(* Logix 5000 project; controller cal1615 1756-L62 rev 20.11; software revision 20.05; part 30 of 81 *)
(* tags used below, declared in another part *)
   FAULT : BOOL;   // Fault AFI
   HMI : BOOL;   // AFI HMI
   p01r09_pb_global_reset : BOOL;   // System Modes PB: Global Fault Reset
   p13_ai_exhaust_amps : REAL;   // Zone 3 Analog Input Exhaust Fan Amps
   p13_ai_exhaust_hz : REAL;   // Zone 3 Analog Input Exhaust Fan HZ
   p13_ai_exhaust_pct : REAL;   // Zone 3 Analog Input Exhaust Fan PCT
   p13_ai_exhaust_rpm : REAL;   // Zone 3 Analog Input Exhaust Fan RPM
   p13_ai_recirc_amps : REAL;   // Zone 3 Analog Input Recirc Fan Amps
   p13_ai_recirc_hz : REAL;   // Zone 3 Analog Input Supply Fan HZ
   p13_ai_recirc_pct : REAL;   // Zone 3 Analog Input Recirc Fan PCT
   p13_ai_recirc_rpm : REAL;   // Zone 3 Analog Input Recirc Fan RPM
   p13_ai_tc01 : REAL;   // Zone 3 Analog Input Control Thermocouple 1
   p13_ai_tc02 : REAL;   // Zone 3 Analog Input Control Thermocouple 2
   p13_ao_cv : REAL;   // Zone 3 Analog Output Control Valve
   p13_ao_exhaust_selected_speed : REAL;   // Zone 3 Analog Output Exhaust Fan VFD Selected Speed
   p13_ao_recirc_selected_speed : REAL;   // Zone 3 Analog Output Recirc Fan VFD Selected Speed
   p13_di_recirc : acs800_di_normal;   // Zone 3 Digital Inputs Recirc Fan
   p13_dint_to_hmi : DINT[16];   // Zone 3 Temperature Control VFDs On
   p13_param_fast_to_soak : REAL;   // Zone 3 Parameter Fast to Soak Control
   p13_param_lfl_hhl : REAL;   // Zone 3 Parameter High High Lower Flash Limit
   p13_param_lfl_hl : REAL;   // Zone 3 Parameter High LFL Limit
   p13_param_pid1_ff : REAL;   // Zone 3 Parameter Fast PID Bias
   p13_param_pid1_kd : REAL;   // Zone 3 Parameter Fast PID Derivative Gain
   p13_param_pid1_ki : REAL;   // Zone 3 Parameter Fast PID Integral Gain
   p13_param_pid1_kp : REAL;   // Zone 3 Parameter Fast PID Proportional Gain
   p13_param_pid2_ff : REAL;   // Zone 3 Parameter Auto PID Bias
   p13_param_pid2_kd : REAL;   // Zone 3 Parameter Auto PID Derivative Gain
   p13_param_pid2_ki : REAL;   // Zone 3 Parameter Auto PID Integral Gain
   p13_param_pid2_kp : REAL;   // Zone 3 Parameter Auto PID Proportional Gain
   p13_param_shutdown_temp : REAL;   // Zone 3 Parameter Zone Shutdown Temperature
   p13_param_soak_to_fast : REAL;   // Zone 3 Parameter Soak to Fast Control
   p13_param_tc01_dev : REAL;   // Zone 3 Parameter Oven Temperature Deviation from Setpoint
   p13_param_tc01_hl : REAL;   // Zone 3 Parameter Process Air High Limit
   p13_param_tc01z : REAL;   // Zone 3 Parameter Process Temperature Zero Offset
   p13_param_tc02z : REAL;   // Zone 3 Parameter SupplyTemperature Zero Offset
   p13_param_zone_pressure : REAL;   // Zone 3 Parameter High Pressure LImit
   p13_real_to_hmi : REAL[112];   // Zone 3 Real to HMI
   p13r01 : routine;   // Zone 3 Main
   p13r05 : routine;   // Zone 3 Dint to HMI
   p13r05_recirc_status : DINT;
   p13r05_timer_fault : TIMER[4];   // Zone 3 Dint to HMI Fault Delay
   p13r05_timer_warning : TIMER[4];   // Zone 3 Dint to HMI Warning Delay
   p13r06 : routine;   // Zone 3 Real to HMI
   p13r06_timer_fault : TIMER[4];   // Zone 3 Real to HMI Fault Delay
   p13r06_timer_warning : TIMER[4];   // Zone 3 Real to HMI Warning Delay
   p13r07 : routine;   // Zone 3 Alarms
   p13r07_timer_fault : TIMER[4];   // Zone 3 Alarms Fault Delay
   p13r07_timer_warning : TIMER[4];   // Zone 3 Alarms Warning Delay
   p13r08 : routine;   // Zone 3 Warnings
   p13r08_timer_fault : TIMER[4];   // Zone 3 Warnings Fault Delay
   p13r08_timer_warning : TIMER[4];   // Zone 3 Warnings Warning Delay
   p13r20 : routine;   // Zone 3 Temp Sequence
   p13r30 : routine;   // Zone 3 Temperature Control
   p13r30_cv_man_sp : REAL;   // Zone 3 Temperature Control Manual Heat Control Valve Setpoint
   p13r30_pid_temp_pv : REAL;   // Zone 3 Temperature Control PID Process Value
   p13r30_pid_temp_sp : REAL;   // Zone 3 Temperature Control PID Temperature Control Setpoint
   p13r31 : routine;   // Zone 3 Exhaust VFD
   p13r32 : routine;   // Zone 3 Recirc VFD
   p13r32_vfd_stopped : BOOL;   // Zone 3 Recirc VFD VFD Stopped
(* P13_Zone_3, continued *)

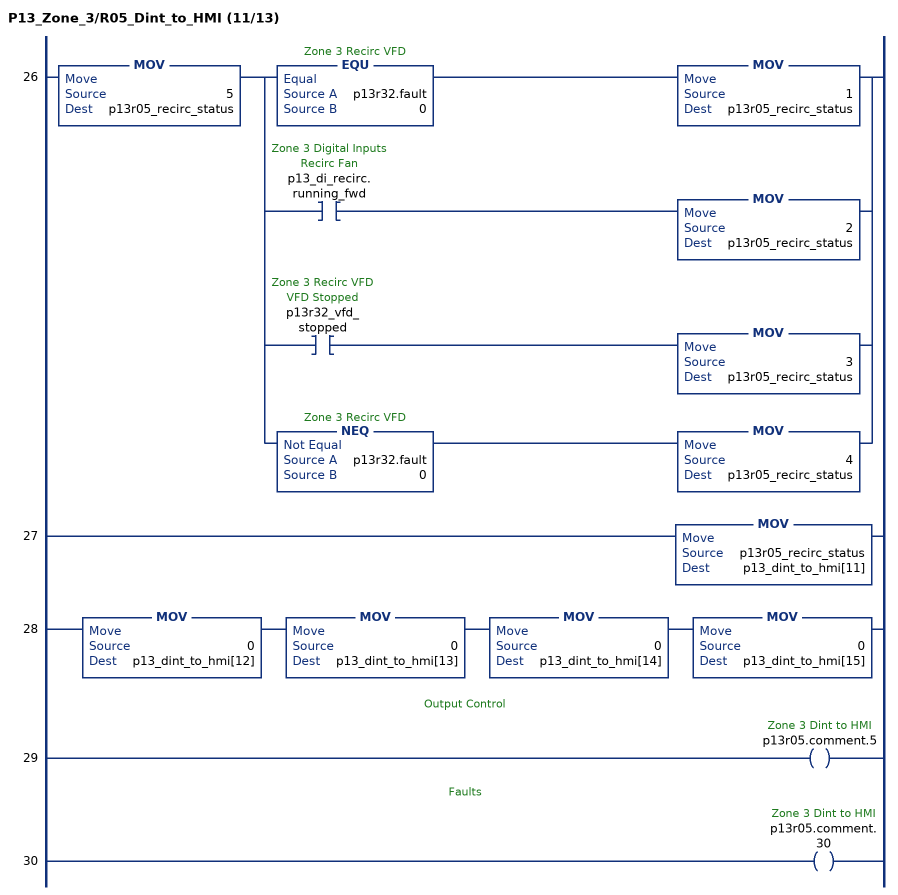
   [picture p524: P13_Zone_3/R05_Dint_to_HMI rungs 26-30]
   26: MOV(5,p13r05_recirc_status)[EQU(p13r32.fault,0) MOV(1,p13r05_recirc_status) ,XIC(p13_di_recirc.running_fwd) MOV(2,p13r05_recirc_status) ,XIC(p13r32_vfd_stopped) MOV(3,p13r05_recirc_status) ,NEQ(p13r32.fault,0) MOV(4,p13r05_recirc_status) ];
   27: MOV(p13r05_recirc_status,p13_dint_to_hmi[11]);
   28: MOV(0,p13_dint_to_hmi[12])MOV(0,p13_dint_to_hmi[13])MOV(0,p13_dint_to_hmi[14])MOV(0,p13_dint_to_hmi[15]);
   // Output Control
   29: OTE(p13r05.comment.5);
   // Faults
   30: OTE(p13r05.comment.30);
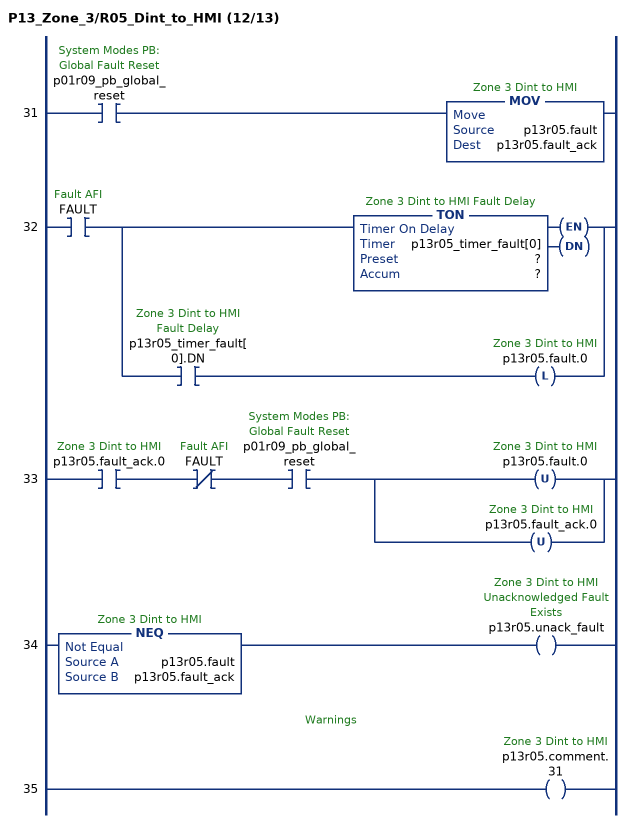
   31: XIC(p01r09_pb_global_reset)MOV(p13r05.fault,p13r05.fault_ack);
   32: XIC(FAULT)[TON(p13r05_timer_fault[0],?,?) ,XIC(p13r05_timer_fault[0].DN) OTL(p13r05.fault.0) ];
   33: XIC(p13r05.fault_ack.0)XIO(FAULT)XIC(p01r09_pb_global_reset)[OTU(p13r05.fault.0) ,OTU(p13r05.fault_ack.0) ];
   34: NEQ(p13r05.fault,p13r05.fault_ack)OTE(p13r05.unack_fault);
   // Warnings
   35: OTE(p13r05.comment.31);
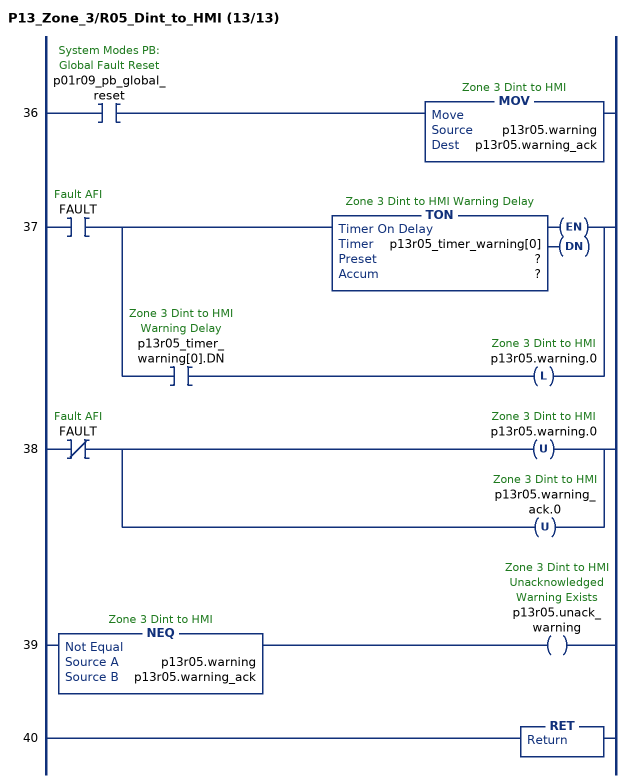
   36: XIC(p01r09_pb_global_reset)MOV(p13r05.warning,p13r05.warning_ack);
   37: XIC(FAULT)[TON(p13r05_timer_warning[0],?,?) ,XIC(p13r05_timer_warning[0].DN) OTL(p13r05.warning.0) ];
   38: XIO(FAULT)[OTU(p13r05.warning.0) ,OTU(p13r05.warning_ack.0) ];
   39: NEQ(p13r05.warning,p13r05.warning_ack)OTE(p13r05.unack_warning);
   40: RET();
END_ROUTINE

ROUTINE R06_Real_to_HMI   (* ladder *)
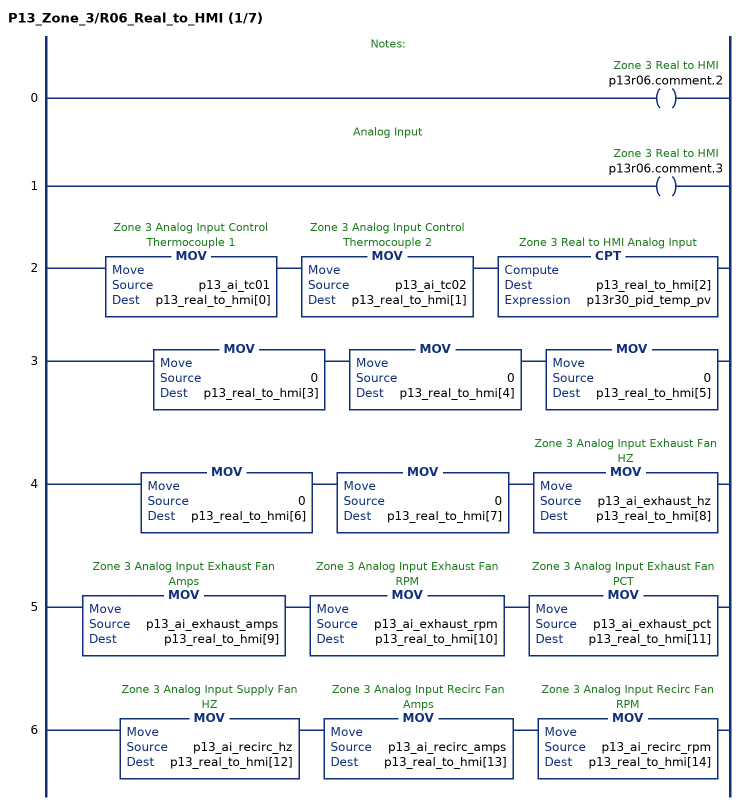
   // Notes:
   0: OTE(p13r06.comment.2);
   // Analog Input
   1: OTE(p13r06.comment.3);
   2: MOV(p13_ai_tc01,p13_real_to_hmi[0])MOV(p13_ai_tc02,p13_real_to_hmi[1])CPT(p13_real_to_hmi[2],p13r30_pid_temp_pv);
   3: MOV(0,p13_real_to_hmi[3])MOV(0,p13_real_to_hmi[4])MOV(0,p13_real_to_hmi[5]);
   4: MOV(0,p13_real_to_hmi[6])MOV(0,p13_real_to_hmi[7])MOV(p13_ai_exhaust_hz,p13_real_to_hmi[8]);
   5: MOV(p13_ai_exhaust_amps,p13_real_to_hmi[9])MOV(p13_ai_exhaust_rpm,p13_real_to_hmi[10])MOV(p13_ai_exhaust_pct,p13_real_to_hmi[11]);
   6: MOV(p13_ai_recirc_hz,p13_real_to_hmi[12])MOV(p13_ai_recirc_amps,p13_real_to_hmi[13])MOV(p13_ai_recirc_rpm,p13_real_to_hmi[14]);
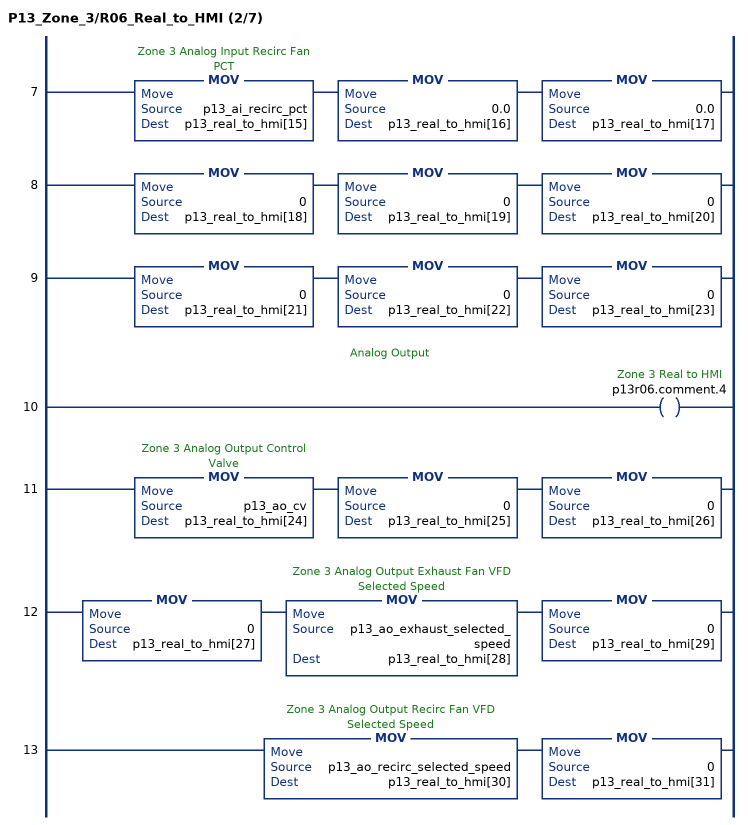
   7: MOV(p13_ai_recirc_pct,p13_real_to_hmi[15])MOV(0.0,p13_real_to_hmi[16])MOV(0.0,p13_real_to_hmi[17]);
   8: MOV(0,p13_real_to_hmi[18])MOV(0,p13_real_to_hmi[19])MOV(0,p13_real_to_hmi[20]);
   9: MOV(0,p13_real_to_hmi[21])MOV(0,p13_real_to_hmi[22])MOV(0,p13_real_to_hmi[23]);
   // Analog Output
   10: OTE(p13r06.comment.4);
   11: MOV(p13_ao_cv,p13_real_to_hmi[24])MOV(0,p13_real_to_hmi[25])MOV(0,p13_real_to_hmi[26]);
   12: MOV(0,p13_real_to_hmi[27])MOV(p13_ao_exhaust_selected_speed,p13_real_to_hmi[28])MOV(0,p13_real_to_hmi[29]);
   13: MOV(p13_ao_recirc_selected_speed,p13_real_to_hmi[30])MOV(0,p13_real_to_hmi[31]);
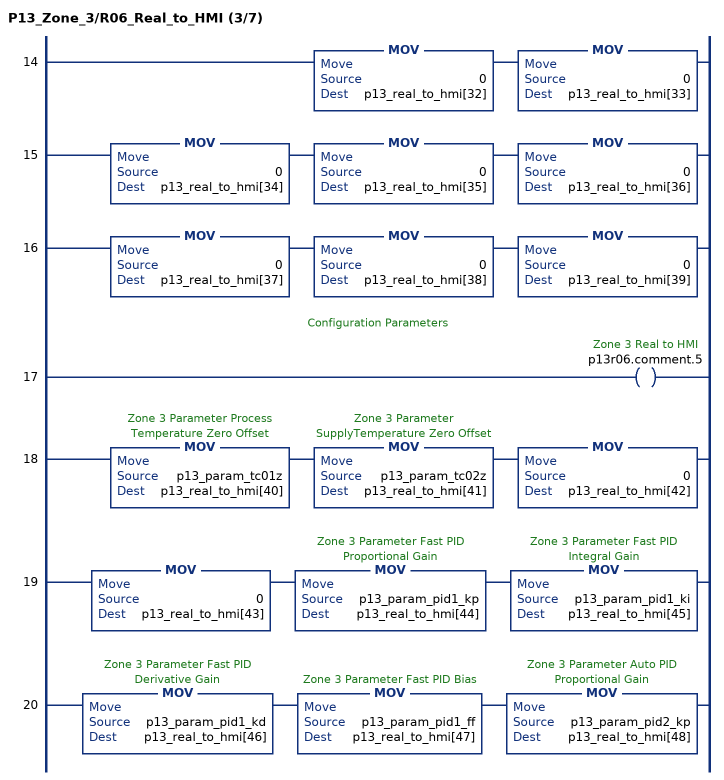
   14: MOV(0,p13_real_to_hmi[32])MOV(0,p13_real_to_hmi[33]);
   15: MOV(0,p13_real_to_hmi[34])MOV(0,p13_real_to_hmi[35])MOV(0,p13_real_to_hmi[36]);
   16: MOV(0,p13_real_to_hmi[37])MOV(0,p13_real_to_hmi[38])MOV(0,p13_real_to_hmi[39]);
   // Configuration Parameters
   17: OTE(p13r06.comment.5);
   18: MOV(p13_param_tc01z,p13_real_to_hmi[40])MOV(p13_param_tc02z,p13_real_to_hmi[41])MOV(0,p13_real_to_hmi[42]);
   19: MOV(0,p13_real_to_hmi[43])MOV(p13_param_pid1_kp,p13_real_to_hmi[44])MOV(p13_param_pid1_ki,p13_real_to_hmi[45]);
   20: MOV(p13_param_pid1_kd,p13_real_to_hmi[46])MOV(p13_param_pid1_ff,p13_real_to_hmi[47])MOV(p13_param_pid2_kp,p13_real_to_hmi[48]);
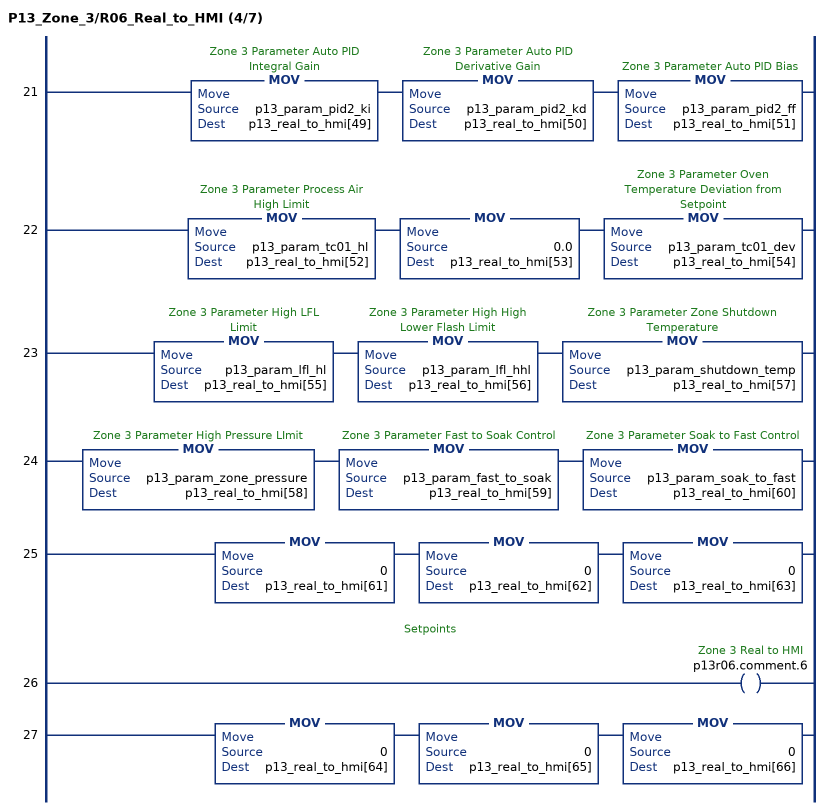
   21: MOV(p13_param_pid2_ki,p13_real_to_hmi[49])MOV(p13_param_pid2_kd,p13_real_to_hmi[50])MOV(p13_param_pid2_ff,p13_real_to_hmi[51]);
   22: MOV(p13_param_tc01_hl,p13_real_to_hmi[52])MOV(0.0,p13_real_to_hmi[53])MOV(p13_param_tc01_dev,p13_real_to_hmi[54]);
   23: MOV(p13_param_lfl_hl,p13_real_to_hmi[55])MOV(p13_param_lfl_hhl,p13_real_to_hmi[56])MOV(p13_param_shutdown_temp,p13_real_to_hmi[57]);
   24: MOV(p13_param_zone_pressure,p13_real_to_hmi[58])MOV(p13_param_fast_to_soak,p13_real_to_hmi[59])MOV(p13_param_soak_to_fast,p13_real_to_hmi[60]);
   25: MOV(0,p13_real_to_hmi[61])MOV(0,p13_real_to_hmi[62])MOV(0,p13_real_to_hmi[63]);
   // Setpoints
   26: OTE(p13r06.comment.6);
   27: MOV(0,p13_real_to_hmi[64])MOV(0,p13_real_to_hmi[65])MOV(0,p13_real_to_hmi[66]);
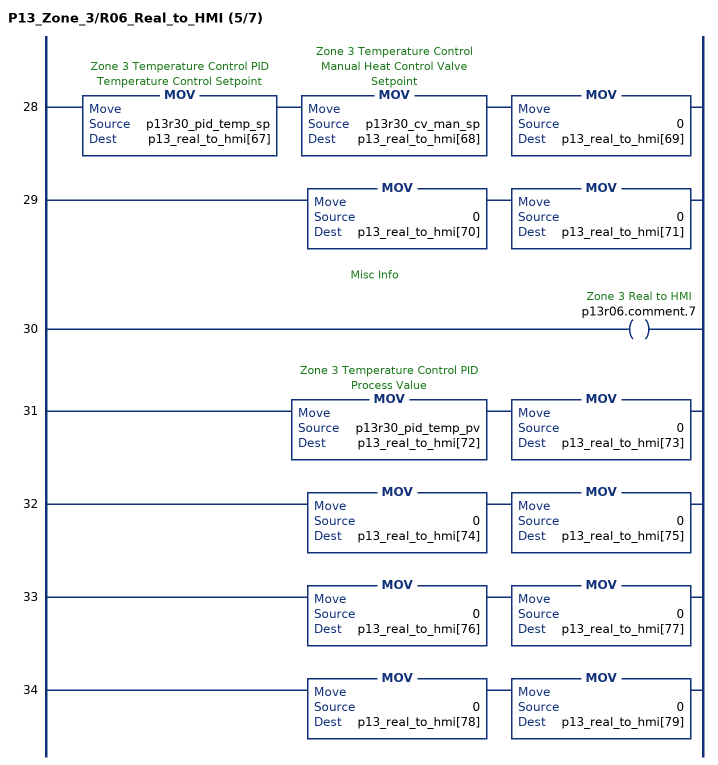
   28: MOV(p13r30_pid_temp_sp,p13_real_to_hmi[67])MOV(p13r30_cv_man_sp,p13_real_to_hmi[68])MOV(0,p13_real_to_hmi[69]);
   29: MOV(0,p13_real_to_hmi[70])MOV(0,p13_real_to_hmi[71]);
   // Misc Info
   30: OTE(p13r06.comment.7);
   31: MOV(p13r30_pid_temp_pv,p13_real_to_hmi[72])MOV(0,p13_real_to_hmi[73]);
   32: MOV(0,p13_real_to_hmi[74])MOV(0,p13_real_to_hmi[75]);
   33: MOV(0,p13_real_to_hmi[76])MOV(0,p13_real_to_hmi[77]);
   34: MOV(0,p13_real_to_hmi[78])MOV(0,p13_real_to_hmi[79]);
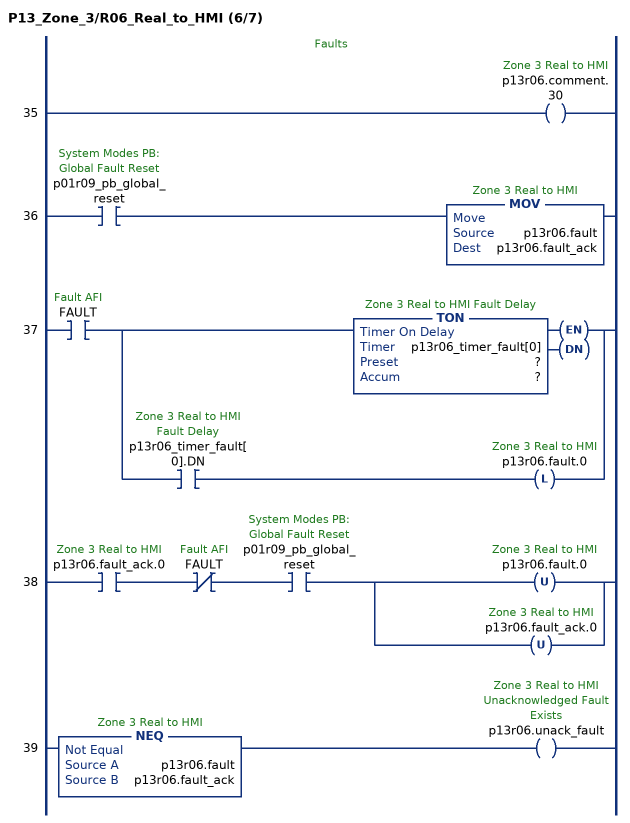
   // Faults
   35: OTE(p13r06.comment.30);
   36: XIC(p01r09_pb_global_reset)MOV(p13r06.fault,p13r06.fault_ack);
   37: XIC(FAULT)[TON(p13r06_timer_fault[0],?,?) ,XIC(p13r06_timer_fault[0].DN) OTL(p13r06.fault.0) ];
   38: XIC(p13r06.fault_ack.0)XIO(FAULT)XIC(p01r09_pb_global_reset)[OTU(p13r06.fault.0) ,OTU(p13r06.fault_ack.0) ];
   39: NEQ(p13r06.fault,p13r06.fault_ack)OTE(p13r06.unack_fault);
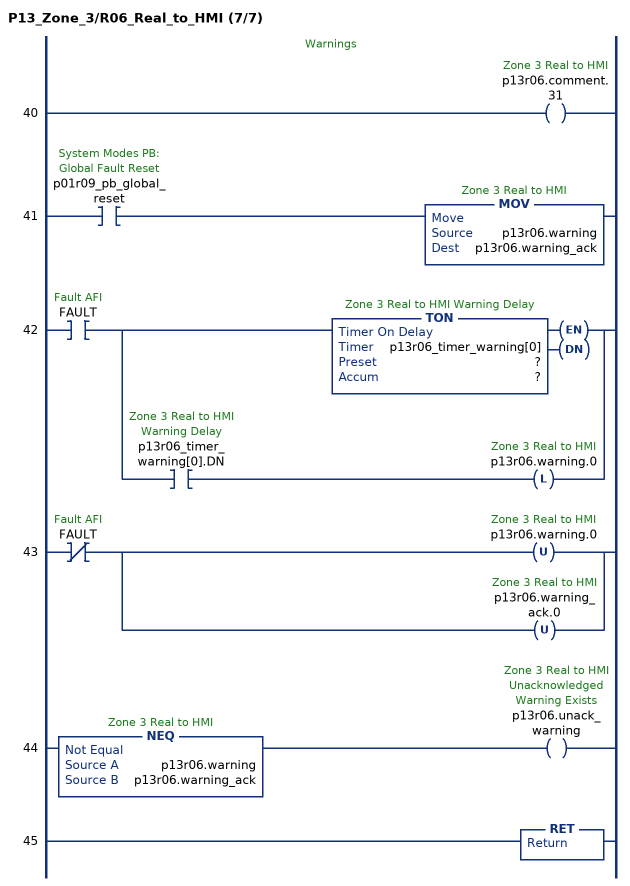
   // Warnings
   40: OTE(p13r06.comment.31);
   41: XIC(p01r09_pb_global_reset)MOV(p13r06.warning,p13r06.warning_ack);
   42: XIC(FAULT)[TON(p13r06_timer_warning[0],?,?) ,XIC(p13r06_timer_warning[0].DN) OTL(p13r06.warning.0) ];
   43: XIO(FAULT)[OTU(p13r06.warning.0) ,OTU(p13r06.warning_ack.0) ];
   44: NEQ(p13r06.warning,p13r06.warning_ack)OTE(p13r06.unack_warning);
   45: RET();
END_ROUTINE

ROUTINE R07_Alarms   (* ladder *)
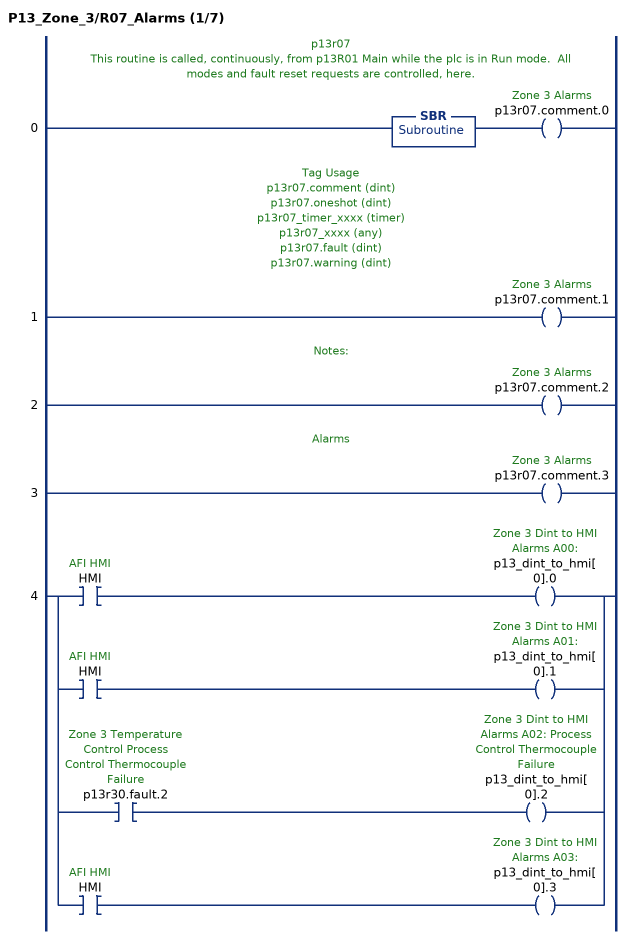
   // p13r07
   // This routine is called, continuously, from p13R01 Main while the plc is in Run mode.  All modes and fault reset requests are controlled, here.
   0: SBR()OTE(p13r07.comment.0);
   // Tag Usage
   // p13r07.comment (dint)
   // p13r07.oneshot (dint)
   // p13r07_timer_xxxx (timer)
   // p13r07_xxxx (any)
   // p13r07.fault (dint)
   // p13r07.warning (dint)
   1: OTE(p13r07.comment.1);
   // Notes:
   2: OTE(p13r07.comment.2);
   // Alarms
   3: OTE(p13r07.comment.3);
   4: [XIC(HMI) OTE(p13_dint_to_hmi[0].0) ,XIC(HMI) OTE(p13_dint_to_hmi[0].1) ,XIC(p13r30.fault.2) OTE(p13_dint_to_hmi[0].2) ,XIC(HMI) OTE(p13_dint_to_hmi[0].3) ];
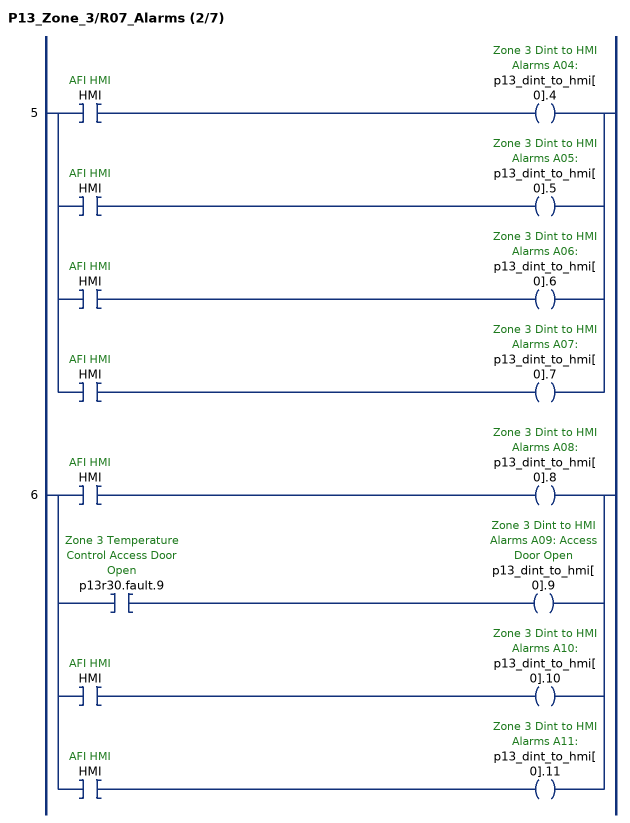
   5: [XIC(HMI) OTE(p13_dint_to_hmi[0].4) ,XIC(HMI) OTE(p13_dint_to_hmi[0].5) ,XIC(HMI) OTE(p13_dint_to_hmi[0].6) ,XIC(HMI) OTE(p13_dint_to_hmi[0].7) ];
   6: [XIC(HMI) OTE(p13_dint_to_hmi[0].8) ,XIC(p13r30.fault.9) OTE(p13_dint_to_hmi[0].9) ,XIC(HMI) OTE(p13_dint_to_hmi[0].10) ,XIC(HMI) OTE(p13_dint_to_hmi[0].11) ];
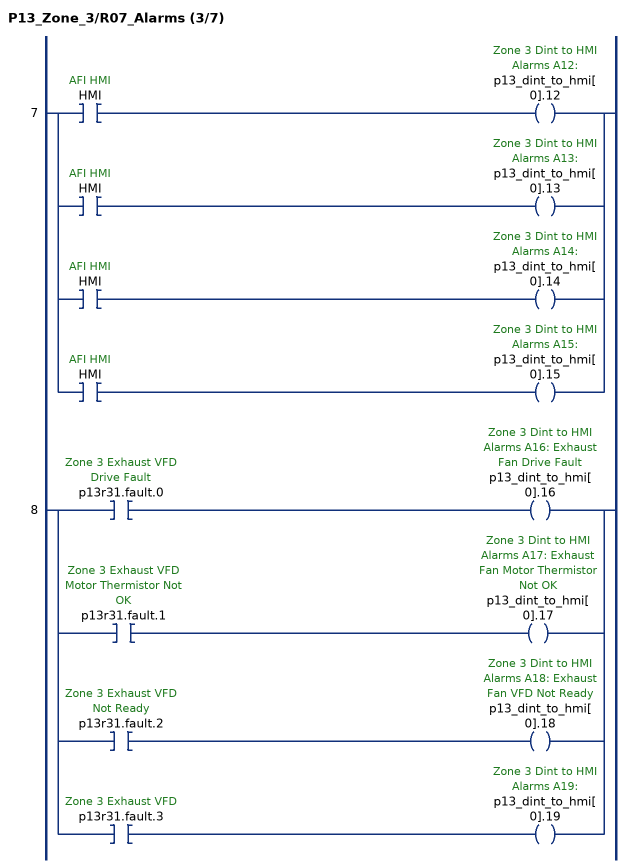
   7: [XIC(HMI) OTE(p13_dint_to_hmi[0].12) ,XIC(HMI) OTE(p13_dint_to_hmi[0].13) ,XIC(HMI) OTE(p13_dint_to_hmi[0].14) ,XIC(HMI) OTE(p13_dint_to_hmi[0].15) ];
   8: [XIC(p13r31.fault.0) OTE(p13_dint_to_hmi[0].16) ,XIC(p13r31.fault.1) OTE(p13_dint_to_hmi[0].17) ,XIC(p13r31.fault.2) OTE(p13_dint_to_hmi[0].18) ,XIC(p13r31.fault.3) OTE(p13_dint_to_hmi[0].19) ];
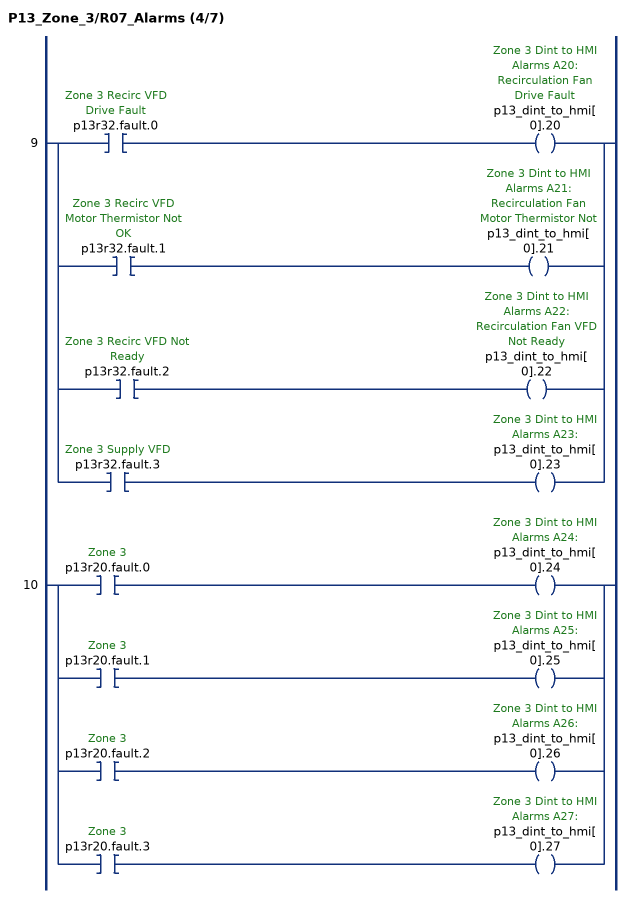
   9: [XIC(p13r32.fault.0) OTE(p13_dint_to_hmi[0].20) ,XIC(p13r32.fault.1) OTE(p13_dint_to_hmi[0].21) ,XIC(p13r32.fault.2) OTE(p13_dint_to_hmi[0].22) ,XIC(p13r32.fault.3) OTE(p13_dint_to_hmi[0].23) ];
   10: [XIC(p13r20.fault.0) OTE(p13_dint_to_hmi[0].24) ,XIC(p13r20.fault.1) OTE(p13_dint_to_hmi[0].25) ,XIC(p13r20.fault.2) OTE(p13_dint_to_hmi[0].26) ,XIC(p13r20.fault.3) OTE(p13_dint_to_hmi[0].27) ];
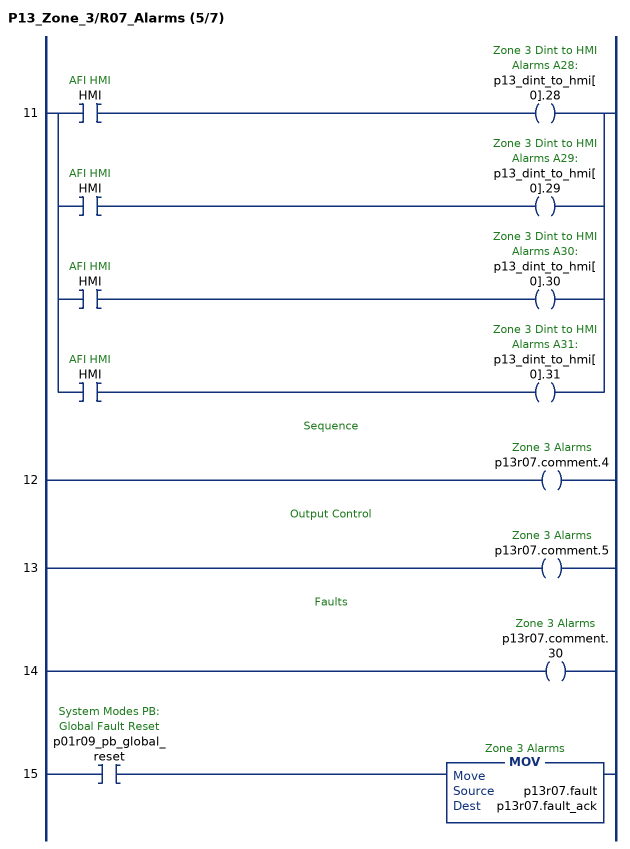
   11: [XIC(HMI) OTE(p13_dint_to_hmi[0].28) ,XIC(HMI) OTE(p13_dint_to_hmi[0].29) ,XIC(HMI) OTE(p13_dint_to_hmi[0].30) ,XIC(HMI) OTE(p13_dint_to_hmi[0].31) ];
   // Sequence
   12: OTE(p13r07.comment.4);
   // Output Control
   13: OTE(p13r07.comment.5);
   // Faults
   14: OTE(p13r07.comment.30);
   15: XIC(p01r09_pb_global_reset)MOV(p13r07.fault,p13r07.fault_ack);
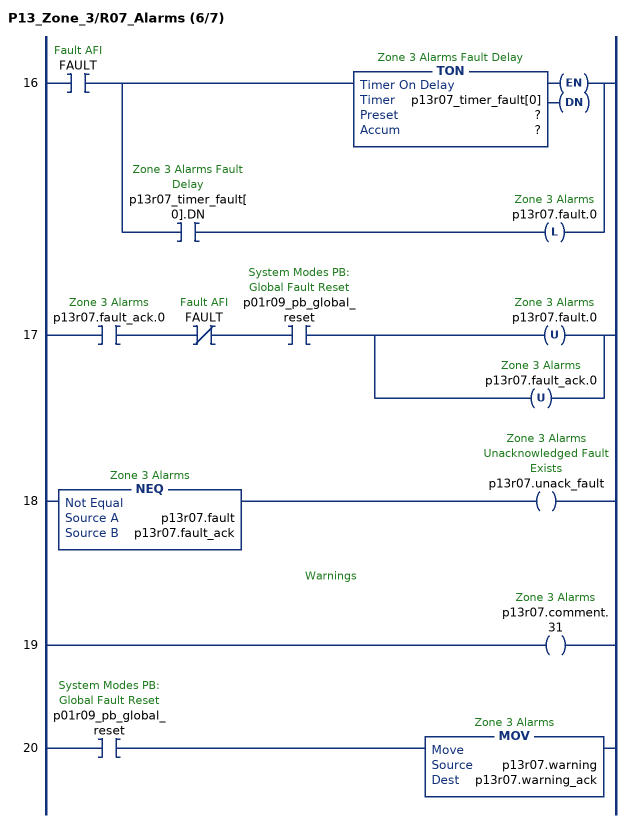
   16: XIC(FAULT)[TON(p13r07_timer_fault[0],?,?) ,XIC(p13r07_timer_fault[0].DN) OTL(p13r07.fault.0) ];
   17: XIC(p13r07.fault_ack.0)XIO(FAULT)XIC(p01r09_pb_global_reset)[OTU(p13r07.fault.0) ,OTU(p13r07.fault_ack.0) ];
   18: NEQ(p13r07.fault,p13r07.fault_ack)OTE(p13r07.unack_fault);
   // Warnings
   19: OTE(p13r07.comment.31);
   20: XIC(p01r09_pb_global_reset)MOV(p13r07.warning,p13r07.warning_ack);
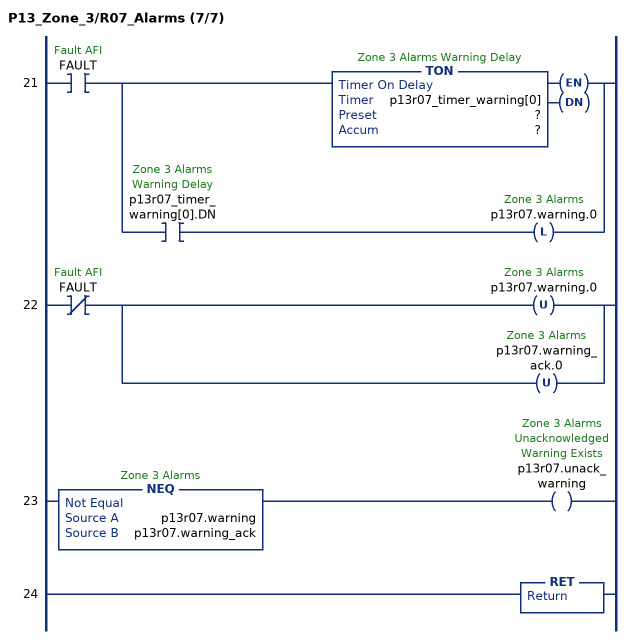
   21: XIC(FAULT)[TON(p13r07_timer_warning[0],?,?) ,XIC(p13r07_timer_warning[0].DN) OTL(p13r07.warning.0) ];
   22: XIO(FAULT)[OTU(p13r07.warning.0) ,OTU(p13r07.warning_ack.0) ];
   23: NEQ(p13r07.warning,p13r07.warning_ack)OTE(p13r07.unack_warning);
   24: RET();
END_ROUTINE

ROUTINE R08_Warnings   (* ladder *)
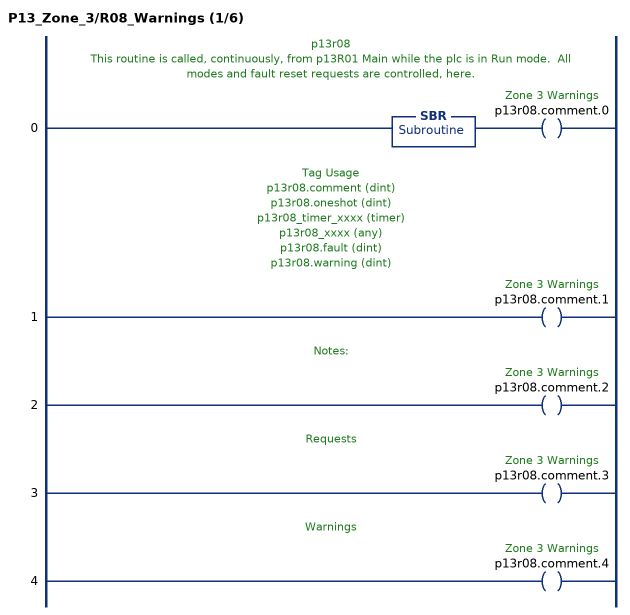
   // p13r08
   // This routine is called, continuously, from p13R01 Main while the plc is in Run mode.  All modes and fault reset requests are controlled, here.
   0: SBR()OTE(p13r08.comment.0);
   // Tag Usage
   // p13r08.comment (dint)
   // p13r08.oneshot (dint)
   // p13r08_timer_xxxx (timer)
   // p13r08_xxxx (any)
   // p13r08.fault (dint)
   // p13r08.warning (dint)
   1: OTE(p13r08.comment.1);
   // Notes:
   2: OTE(p13r08.comment.2);
   // Requests
   3: OTE(p13r08.comment.3);
   // Warnings
   4: OTE(p13r08.comment.4);
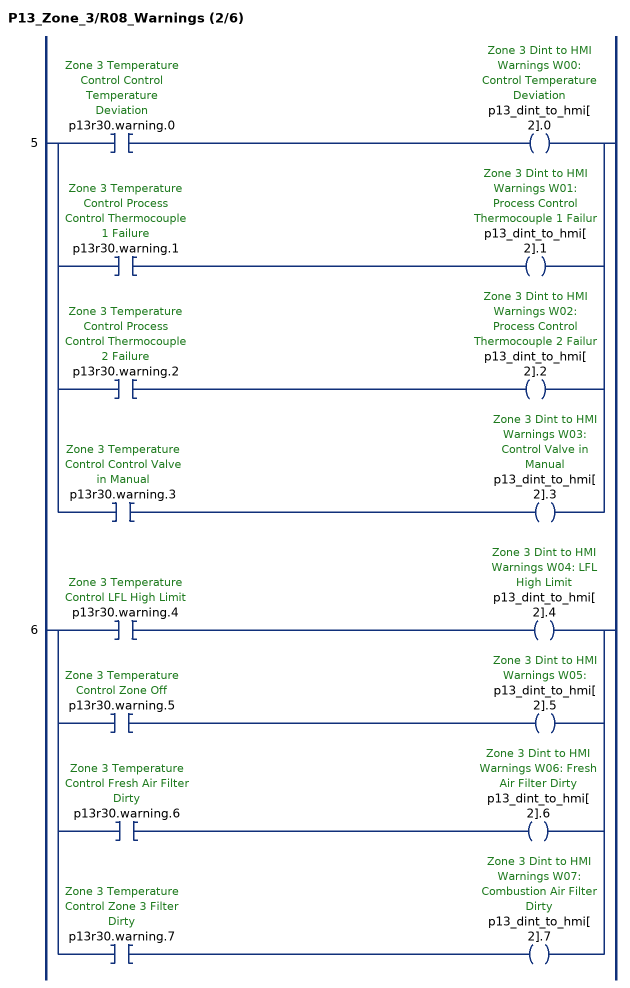
   5: [XIC(p13r30.warning.0) OTE(p13_dint_to_hmi[2].0) ,XIC(p13r30.warning.1) OTE(p13_dint_to_hmi[2].1) ,XIC(p13r30.warning.2) OTE(p13_dint_to_hmi[2].2) ,XIC(p13r30.warning.3) OTE(p13_dint_to_hmi[2].3) ];
   6: [XIC(p13r30.warning.4) OTE(p13_dint_to_hmi[2].4) ,XIC(p13r30.warning.5) OTE(p13_dint_to_hmi[2].5) ,XIC(p13r30.warning.6) OTE(p13_dint_to_hmi[2].6) ,XIC(p13r30.warning.7) OTE(p13_dint_to_hmi[2].7) ];
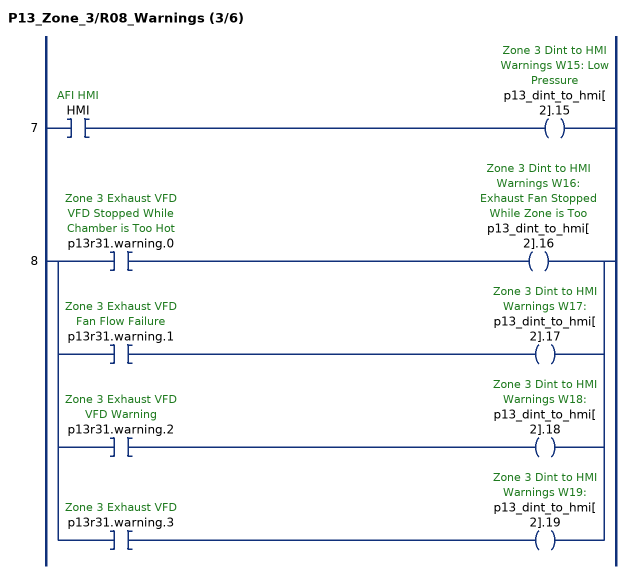
   7: XIC(HMI)OTE(p13_dint_to_hmi[2].15);
   8: [XIC(p13r31.warning.0) OTE(p13_dint_to_hmi[2].16) ,XIC(p13r31.warning.1) OTE(p13_dint_to_hmi[2].17) ,XIC(p13r31.warning.2) OTE(p13_dint_to_hmi[2].18) ,XIC(p13r31.warning.3) OTE(p13_dint_to_hmi[2].19) ];
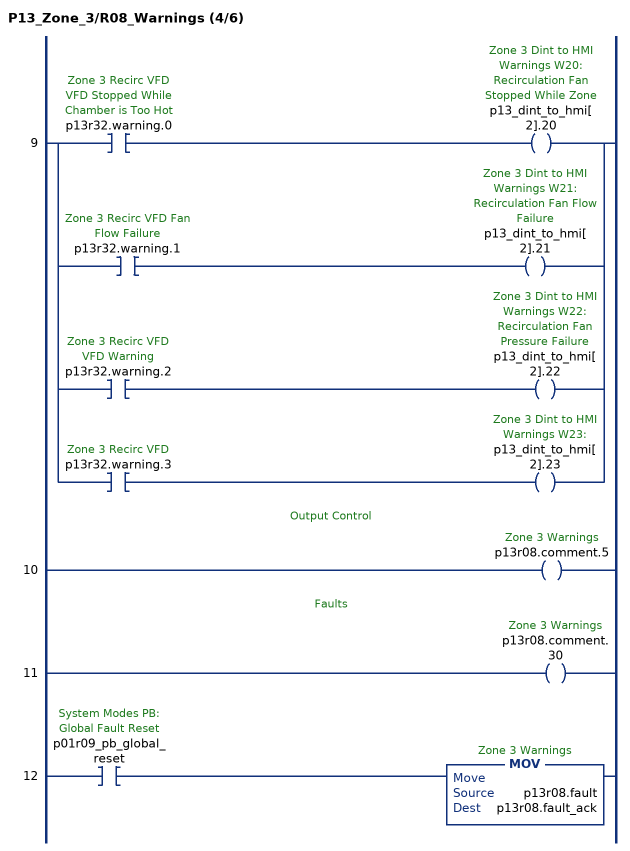
   9: [XIC(p13r32.warning.0) OTE(p13_dint_to_hmi[2].20) ,XIC(p13r32.warning.1) OTE(p13_dint_to_hmi[2].21) ,XIC(p13r32.warning.2) OTE(p13_dint_to_hmi[2].22) ,XIC(p13r32.warning.3) OTE(p13_dint_to_hmi[2].23) ];
   // Output Control
   10: OTE(p13r08.comment.5);
   // Faults
   11: OTE(p13r08.comment.30);
   12: XIC(p01r09_pb_global_reset)MOV(p13r08.fault,p13r08.fault_ack);
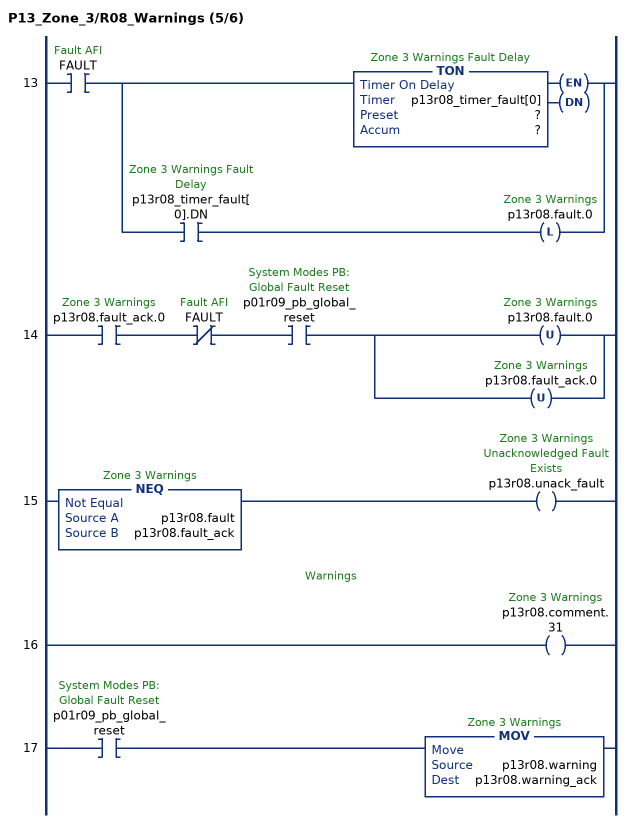
   13: XIC(FAULT)[TON(p13r08_timer_fault[0],?,?) ,XIC(p13r08_timer_fault[0].DN) OTL(p13r08.fault.0) ];
   14: XIC(p13r08.fault_ack.0)XIO(FAULT)XIC(p01r09_pb_global_reset)[OTU(p13r08.fault.0) ,OTU(p13r08.fault_ack.0) ];
   15: NEQ(p13r08.fault,p13r08.fault_ack)OTE(p13r08.unack_fault);
   // Warnings
   16: OTE(p13r08.comment.31);
   17: XIC(p01r09_pb_global_reset)MOV(p13r08.warning,p13r08.warning_ack);
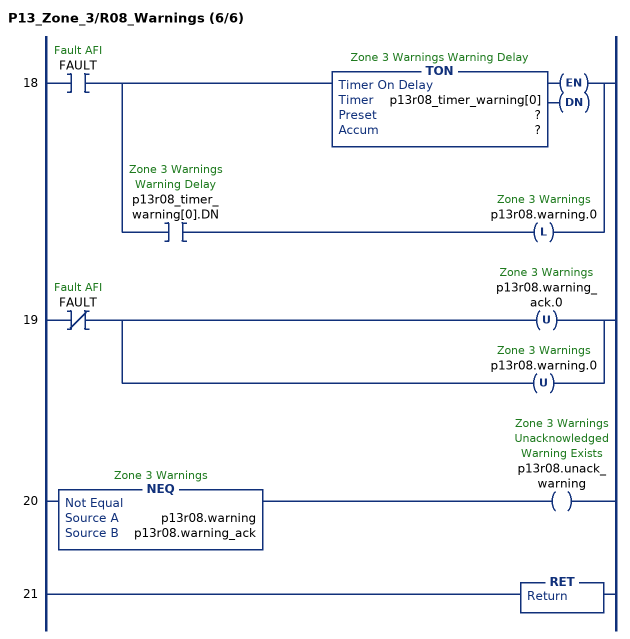
   18: XIC(FAULT)[TON(p13r08_timer_warning[0],?,?) ,XIC(p13r08_timer_warning[0].DN) OTL(p13r08.warning.0) ];
   19: XIO(FAULT)[OTU(p13r08.warning_ack.0) ,OTU(p13r08.warning.0) ];
   20: NEQ(p13r08.warning,p13r08.warning_ack)OTE(p13r08.unack_warning);
   21: RET();
END_ROUTINE
